Fanuc KAREL source: kc00010.KL

-- PROVISIONAL review KL for V940-1; original PC SHA256 8fb04647ad982aca0350fa127ea5d831413367fc5437d2bdf128436cbf9e4c05
-- Incomplete behavior may be omitted. Consult companion uncertainty JSON. Do not deploy.
PROGRAM KC00010
%NOLOCKGROUP
BEGIN
  -- V9_ZERO_TABLE_METADATA_HINT layout=0002_ascii; no indexed target words; source/name/runtime held
  -- UNRESOLVED_PC offsets 5-27; opcodes 27,22,1C,31,23
  -- UNRESOLVED_PC offsets 32-36; opcodes 7F
END KC00010
